INTERFACE I_MotionInterlocksCommon  EXTENDS I_Error

METHOD DriveCommands
VAR_INPUT
	Enable: BOOL;
	NewMoveReq : BOOL;
END_VAR
END_METHOD

PROPERTY HardwareEnable : BOOL
GET
END_GET
END_PROPERTY

PROPERTY MoveOk : BOOL
GET
END_GET
END_PROPERTY

PROPERTY PowerEnabled : BOOL
GET
END_GET
END_PROPERTY

METHOD Reset
VAR_INPUT
END_VAR
END_METHOD

PROPERTY UserEnable : BOOL
SET
END_SET
END_PROPERTY

END_INTERFACE

(* stored: Version 1.1.0.1
   Itf I_MotionInterlocksCommon: Id {6906b881-f15f-4df2-99d8-615248381a43}
   Method DriveCommands: Id {b62a5c4b-ba10-475e-b112-d1bdb58ba629}
   Property HardwareEnable: Id {340fc236-f476-43a5-8232-685aab4a5a0e}
   Get Get: Id {8af58745-28c2-4726-b711-8ab5523bc308}
   Property MoveOk: Id {1afd93f7-f2a6-41c4-917d-1b6c9a77ea87}
   Get Get: Id {eb795768-982c-4440-9ee6-002d67c772ee}
   Property PowerEnabled: Id {c51eea5c-413d-4ba5-abaf-3b70155b6bdc}
   Get Get: Id {05bad098-7800-4d94-a94a-923a51852e71}
   Method Reset: Id {cc36a04e-8ae1-4d1a-b6d2-3ef1ada15b9d}
   Property UserEnable: Id {16b82871-fb73-4df5-80f5-08b1172c1b10}
   Set Set: Id {e08ffba2-63ce-4002-9296-5aee47ddb046} *)
